{attribute 'qualified_only'}
{attribute 'strict'}
{attribute 'to_string'}
TYPE E_TemperatureUnit  :
(
   Celsius := 0,
    Fahrenheit := 1,
    Kelvin := 2,
    Rankine := 3
);
END_TYPE

(* stored: Version 1.1.0.1
   DUT E_TemperatureUnit: Id {ebc15123-5807-4bc9-8435-e57b9e4ea996} *)
